TYPE XYParams_typ :
STRUCT
	bUserIncrementStep		: BOOL;
	bUserInfiniteMovement 	: BOOL; 
	nState					: INT;
	nNextState				: INT;
	fVelFactor				: LREAL;
END_STRUCT
END_TYPE

(* stored: Version 1.1.0.1, ProductVersion 3.1.4024.11
   DUT XYParams_typ: Id {96125d31-1a1d-4672-8e3a-7a436b006c4f} *)
